FUNCTION CheckFault : BOOL
VAR_INPUT
	Overload: BOOL;
	MotorTemp: INT;
	
END_VAR
VAR
END_VAR

IF Overload OR MotorTemp > 80 THEN
	CheckFault:=TRUE;
ELSE
	CheckFault:=FALSE;
END_IF

END_FUNCTION

(* stored: Version 1.1.0.1, ProductVersion 3.1.4024.9
   POU CheckFault: Id {6fc24085-08b8-46ad-89b9-b83ba09abd5d}, SpecialFunc None *)
